FUNCTION_BLOCK SS5_ps_v1 (* Composite FB wrapping other FBs *)
  (* Standard: 61499-2 *)
  (* Version 1.0, 2025-07-23, DEVIASH *)
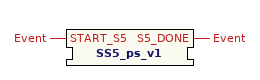
  EVENT_INPUT
    START_S5;
  END_EVENT
  EVENT_OUTPUT
    S5_DONE;
  END_EVENT
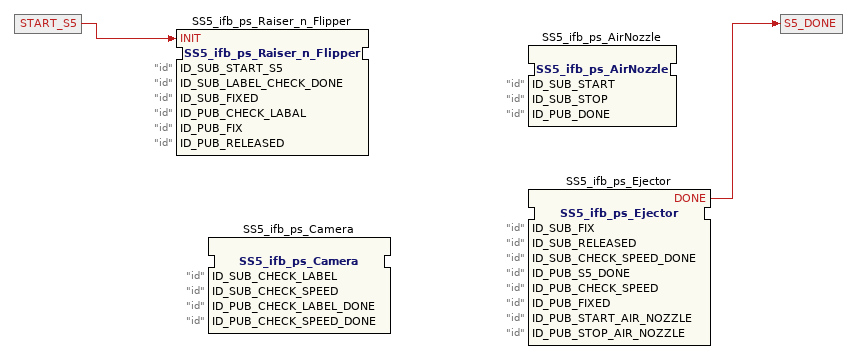
  FBS
    SS5_ifb_ps_AirNozzle : SS5_ifb_ps_AirNozzle(ID_SUB_START := "id", ID_SUB_STOP := "id", ID_PUB_DONE := "id");
    SS5_ifb_ps_Camera : UserLibs::SubStations::SS5::SS5_ifb_ps_Camera(ID_SUB_CHECK_LABEL := "id", ID_SUB_CHECK_SPEED := "id", ID_PUB_CHECK_LABEL_DONE := "id", ID_PUB_CHECK_SPEED_DONE := "id");
    SS5_ifb_ps_Ejector : UserLibs::SubStations::SS5::SS5_ifb_ps_Ejector(ID_SUB_FIX := "id", ID_SUB_RELEASED := "id", ID_SUB_CHECK_SPEED_DONE := "id", ID_PUB_S5_DONE := "id", ID_PUB_CHECK_SPEED := "id", ID_PUB_FIXED := "id", ID_PUB_START_AIR_NOZZLE := "id", ID_PUB_STOP_AIR_NOZZLE := "id");
    SS5_ifb_ps_Raiser_n_Flipper : UserLibs::SubStations::SS5::SS5_ifb_ps_Raiser_n_Flipper(ID_SUB_START_S5 := "id", ID_SUB_LABEL_CHECK_DONE := "id", ID_SUB_FIXED := "id", ID_PUB_CHECK_LABAL := "id", ID_PUB_FIX := "id", ID_PUB_RELEASED := "id");
  END_FBS
  EVENT_CONNECTIONS
    START_S5 TO SS5_ifb_ps_Raiser_n_Flipper.INIT;
    SS5_ifb_ps_Ejector.DONE TO S5_DONE;
  END_CONNECTIONS
END_FUNCTION_BLOCK
